{attribute addProperty BoxType "EL6201-0000-0017"}
{attribute addProperty Id "Slave_1_InputsAT %I*Slave_1_Inputs_412A1CB0811Slave_2_InputsAT %I*Slave_2_Inputs_32ADBE12819Slave_3_InputsAT %I*Slave_3_Inputs_09EFF6788117Slave_4_InputsAT %I*Slave_4_Inputs_CB1B8FCC8125Slave_5_InputsAT %I*Slave_5_Inputs_39F4F5D68133Slave_6_InputsAT %I*Slave_6_Inputs_3F922B488141Slave_7_InputsAT %I*Slave_7_Inputs_634B595D8149Slave_8_InputsAT %I*Slave_8_Inputs_A0929BA58157Slave_9_InputsAT %I*Slave_9_Inputs_7914DDDE8165Slave_10_InputsAT %I*Slave_10_Inputs_7E96E18B8173Slave_11_InputsAT %I*Slave_11_Inputs_E06D80F08181Slave_12_InputsAT %I*Slave_12_Inputs_13FE58598189Slave_13_InputsAT %I*Slave_13_Inputs_5BEA61188197Slave_14_InputsAT %I*Slave_14_Inputs_AC35CC5681105Slave_15_InputsAT %I*Slave_15_Inputs_B7A05B5581113Slave_16_InputsAT %I*Slave_16_Inputs_9C95469381121Slave_17_InputsAT %I*Slave_17_Inputs_FE539A7F81129Slave_18_InputsAT %I*Slave_18_Inputs_FC91B4FB81137Slave_19_InputsAT %I*Slave_19_Inputs_B78CDC4981145Slave_20_InputsAT %I*Slave_20_Inputs_8F92772781153Slave_21_InputsAT %I*Slave_21_Inputs_C9D920AE81161Slave_22_InputsAT %I*Slave_22_Inputs_C661B60D81169Slave_23_InputsAT %I*Slave_23_Inputs_654EBC1781177Slave_24_InputsAT %I*Slave_24_Inputs_B303EEEB81185Slave_25_InputsAT %I*Slave_25_Inputs_8045513C81193Slave_26_InputsAT %I*Slave_26_Inputs_6028C8D081201Slave_27_InputsAT %I*Slave_27_Inputs_02EE143C81209Slave_28_InputsAT %I*Slave_28_Inputs_5387DDDA81217Slave_29_InputsAT %I*Slave_29_Inputs_8F9349FC81225Slave_30_InputsAT %I*Slave_30_Inputs_118BCC7F81233Slave_31_InputsAT %I*Slave_31_Inputs_D646A1A981241"}
{attribute addProperty CRC "1848625427"}
{attribute addProperty SizeInBites "248"}
{attribute addProperty SizeInBytes "31"}
TYPE ASI_Inputs_Device_6E2FC913 :
STRUCT
	{attribute addProperty Name "Slave_1_Inputs"}
	Slave_1_Inputs AT %I* : Slave_1_Inputs_412A1CB0;
	{attribute addProperty Name "Slave_2_Inputs"}
	Slave_2_Inputs AT %I* : Slave_2_Inputs_32ADBE12;
	{attribute addProperty Name "Slave_3_Inputs"}
	Slave_3_Inputs AT %I* : Slave_3_Inputs_09EFF678;
	{attribute addProperty Name "Slave_4_Inputs"}
	Slave_4_Inputs AT %I* : Slave_4_Inputs_CB1B8FCC;
	{attribute addProperty Name "Slave_5_Inputs"}
	Slave_5_Inputs AT %I* : Slave_5_Inputs_39F4F5D6;
	{attribute addProperty Name "Slave_6_Inputs"}
	Slave_6_Inputs AT %I* : Slave_6_Inputs_3F922B48;
	{attribute addProperty Name "Slave_7_Inputs"}
	Slave_7_Inputs AT %I* : Slave_7_Inputs_634B595D;
	{attribute addProperty Name "Slave_8_Inputs"}
	Slave_8_Inputs AT %I* : Slave_8_Inputs_A0929BA5;
	{attribute addProperty Name "Slave_9_Inputs"}
	Slave_9_Inputs AT %I* : Slave_9_Inputs_7914DDDE;
	{attribute addProperty Name "Slave_10_Inputs"}
	Slave_10_Inputs AT %I* : Slave_10_Inputs_7E96E18B;
	{attribute addProperty Name "Slave_11_Inputs"}
	Slave_11_Inputs AT %I* : Slave_11_Inputs_E06D80F0;
	{attribute addProperty Name "Slave_12_Inputs"}
	Slave_12_Inputs AT %I* : Slave_12_Inputs_13FE5859;
	{attribute addProperty Name "Slave_13_Inputs"}
	Slave_13_Inputs AT %I* : Slave_13_Inputs_5BEA6118;
	{attribute addProperty Name "Slave_14_Inputs"}
	Slave_14_Inputs AT %I* : Slave_14_Inputs_AC35CC56;
	{attribute addProperty Name "Slave_15_Inputs"}
	Slave_15_Inputs AT %I* : Slave_15_Inputs_B7A05B55;
	{attribute addProperty Name "Slave_16_Inputs"}
	Slave_16_Inputs AT %I* : Slave_16_Inputs_9C954693;
	{attribute addProperty Name "Slave_17_Inputs"}
	Slave_17_Inputs AT %I* : Slave_17_Inputs_FE539A7F;
	{attribute addProperty Name "Slave_18_Inputs"}
	Slave_18_Inputs AT %I* : Slave_18_Inputs_FC91B4FB;
	{attribute addProperty Name "Slave_19_Inputs"}
	Slave_19_Inputs AT %I* : Slave_19_Inputs_B78CDC49;
	{attribute addProperty Name "Slave_20_Inputs"}
	Slave_20_Inputs AT %I* : Slave_20_Inputs_8F927727;
	{attribute addProperty Name "Slave_21_Inputs"}
	Slave_21_Inputs AT %I* : Slave_21_Inputs_C9D920AE;
	{attribute addProperty Name "Slave_22_Inputs"}
	Slave_22_Inputs AT %I* : Slave_22_Inputs_C661B60D;
	{attribute addProperty Name "Slave_23_Inputs"}
	Slave_23_Inputs AT %I* : Slave_23_Inputs_654EBC17;
	{attribute addProperty Name "Slave_24_Inputs"}
	Slave_24_Inputs AT %I* : Slave_24_Inputs_B303EEEB;
	{attribute addProperty Name "Slave_25_Inputs"}
	Slave_25_Inputs AT %I* : Slave_25_Inputs_8045513C;
	{attribute addProperty Name "Slave_26_Inputs"}
	Slave_26_Inputs AT %I* : Slave_26_Inputs_6028C8D0;
	{attribute addProperty Name "Slave_27_Inputs"}
	Slave_27_Inputs AT %I* : Slave_27_Inputs_02EE143C;
	{attribute addProperty Name "Slave_28_Inputs"}
	Slave_28_Inputs AT %I* : Slave_28_Inputs_5387DDDA;
	{attribute addProperty Name "Slave_29_Inputs"}
	Slave_29_Inputs AT %I* : Slave_29_Inputs_8F9349FC;
	{attribute addProperty Name "Slave_30_Inputs"}
	Slave_30_Inputs AT %I* : Slave_30_Inputs_118BCC7F;
	{attribute addProperty Name "Slave_31_Inputs"}
	Slave_31_Inputs AT %I* : Slave_31_Inputs_D646A1A9;
END_STRUCT
END_TYPE

(* stored: Version 1.2.0.0, ProductVersion 3.1.4024.9
   DUT ASI_Inputs_Device_6E2FC913: Id {0c3d85ad-00b8-4e96-950a-f4d9283dbb4b} *)
